// TIA Portal V16 export
// export: Created 2024-12-03T15:41:44.0286551Z, ExportSetting WithDefaults, DisplayName Totally Integrated Automation Portal, DisplayVersion V16 Update 6, DisplayName TIA Portal Version Control Interface, DisplayVersion V16 Update 2, DisplayName TIA Portal Openness, DisplayVersion V16 Update 6, DisplayName TIA Portal Teamcenter Gateway, DisplayVersion V16, DisplayName SINAMICS Startdrive Advanced, DisplayVersion V16 Update 5, DisplayName SINAMICS Startdrive G130, G150, S120, S150, SINAMICS MV, S210, DisplayVersion V16 Update 5, DisplayName SINAMICS Startdrive G110M, G120, G120C, G120D, G120P, G115D, DisplayVersion V16 Update 5, DisplayName STEP 7 Professional, DisplayVersion V16 Update 6, DisplayName STEP 7 Safety, DisplayVersion V16, DisplayName WinCC Advanced / Unified PC, DisplayVersion V16 Update 6
DATA_BLOCK "CONV_DB"   // DB49
{ S7_Optimized_Access := 'FALSE' }
VERSION : 0.1
// stored: AutoNumber true, DBAccessibleFromOPCUA true, IsOnlyStoredInLoadMemory false, IsWriteProtectedInAS false
   VAR
      empty : "Conveyor_UDT";
      CONV_101 : "Conveyor_UDT";
      CONV_102L : "Conveyor_UDT";
      CONV_102R : "Conveyor_UDT";
      CONV_103L { S7_SetPoint := 'True'} : "Conveyor_UDT";
      CONV_103R { S7_SetPoint := 'True'} : "Conveyor_UDT";
      CONV_104L { S7_SetPoint := 'True'} : "Conveyor_UDT";
      CONV_104R { S7_SetPoint := 'True'} : "Conveyor_UDT";
      CONV_105L { S7_SetPoint := 'True'} : "Conveyor_UDT";
      CONV_105R { S7_SetPoint := 'True'} : "Conveyor_UDT";
      CONV_106R { S7_SetPoint := 'True'} : "Conveyor_UDT";
      CONV_107R { S7_SetPoint := 'True'} : "Conveyor_UDT";
      CONV_108L { S7_SetPoint := 'True'} : "Conveyor_UDT";
      CONV_108R { S7_SetPoint := 'True'} : "Conveyor_UDT";
      CONV_109L { S7_SetPoint := 'True'} : "Conveyor_UDT";
      CONV_109R { S7_SetPoint := 'True'} : "Conveyor_UDT";
      CONV_110L { S7_SetPoint := 'True'} : "Conveyor_UDT";
      CONV_110R { S7_SetPoint := 'True'} : "Conveyor_UDT";
      CONV_111L { S7_SetPoint := 'True'} : "Conveyor_UDT";
      CONV_111R { S7_SetPoint := 'True'} : "Conveyor_UDT";
      CONV_112R { S7_SetPoint := 'True'} : "Conveyor_UDT";
      CONV_113L { S7_SetPoint := 'True'} : "Conveyor_UDT";
      CONV_113R { S7_SetPoint := 'True'} : "Conveyor_UDT";
      CONV_114L { S7_SetPoint := 'True'} : "Conveyor_UDT";
      CONV_114R { S7_SetPoint := 'True'} : "Conveyor_UDT";
      CONV_115L { S7_SetPoint := 'True'} : "Conveyor_UDT";
      CONV_115R { S7_SetPoint := 'True'} : "Conveyor_UDT";
      CONV_201R_BELTS { S7_SetPoint := 'True'} : "Conveyor_UDT";
      CONV_203R_BELTS { S7_SetPoint := 'True'} : "Conveyor_UDT";
      CONV_301R { S7_SetPoint := 'True'} : "Conveyor_UDT";
      CONV_302L { S7_SetPoint := 'True'} : "Conveyor_UDT";
      CONV_302R { S7_SetPoint := 'True'} : "Conveyor_UDT";
      CONV_303L { S7_SetPoint := 'True'} : "Conveyor_UDT";
      CONV_303R { S7_SetPoint := 'True'} : "Conveyor_UDT";
      CONV_304L { S7_SetPoint := 'True'} : "Conveyor_UDT";
      CONV_304R { S7_SetPoint := 'True'} : "Conveyor_UDT";
      CONV_305R { S7_SetPoint := 'True'} : "Conveyor_UDT";
   END_VAR
BEGIN
   CONV_102L.Settings.Direction := TRUE;
   CONV_102L.Settings.Timings.ReceiveDistance := 300.0;
END_DATA_BLOCK
